// TIA Portal V18 export
VAR_GLOBAL   // PLC tag table "Default tag table"
   "AI11.01.01" AT %IW64 : Int;   // AHU NF Перепад тиску повітря (2.40)
   "AI11.01.02" AT %IW66 : Int;   // HS Вихід нагрівача (10.11)
   "DI11.01.01" AT %I0.0 : Bool;   // HS Режим роботи "Зима"
   "DI11.01.02" AT %I0.1 : Bool;   // HS Режим роботи "Авто"
   "DI11.01.03" AT %I0.2 : Bool;   // HS Відмова Котел 1
   "DI11.01.04" AT %I0.3 : Bool;   // HS Відмова Котел 2
   "DI11.01.05" AT %I0.4 : Bool;   // HS Норм. рівень води Котел 1 (10.80)
   "DI11.01.06" AT %I0.5 : Bool;   // HS Низький тиск Котел 1 (10.71)
   "DI11.01.07" AT %I0.6 : Bool;   // HS Високий тиск Котел 1 (10.72)
   "DI11.01.08" AT %I0.7 : Bool;   // HS Норм. рівень води Котел 2 (10.81)
   "DI11.01.09" AT %I1.0 : Bool;   // HS Низький тиск Котел 1 (10.73)
   "DI11.01.10" AT %I1.1 : Bool;   // HS Високий тиск Котел 1 (10.74)
   "DI11.01.11" AT %I1.2 : Bool;
   "DI11.01.12" AT %I1.3 : Bool;
   "DI11.01.13" AT %I1.4 : Bool;
   "DI11.01.14" AT %I1.5 : Bool;
   "DO11.01.01" AT %Q0.0 : Bool;
   "DO11.01.02" AT %Q0.1 : Bool;
   "DO11.01.03" AT %Q0.2 : Bool;
   "DO11.01.04" AT %Q0.3 : Bool;
   "DO11.01.05" AT %Q0.4 : Bool;
   "DO11.01.06" AT %Q0.5 : Bool;
   "DO11.01.07" AT %Q0.6 : Bool;
   "DO11.01.08" AT %Q0.7 : Bool;
   "DO11.01.09" AT %Q1.0 : Bool;
   "DO11.01.10" AT %Q1.1 : Bool;
   "AI11.02.01" AT %IW68 : Int;
   "AI11.02.02" AT %IW70 : Int;
   "AI11.02.03" AT %IW72 : Int;
   "AI11.02.04" AT %IW74 : Int;
   "AI11.02.05" AT %IW76 : Int;
   "AI11.02.06" AT %IW78 : Int;
   "AI11.02.07" AT %IW80 : Int;
   "AI11.02.08" AT %IW82 : Int;
   "AO11.03.01" AT %QW64 : Int;
   "AO11.03.02" AT %QW66 : Int;
   "AO11.03.03" AT %QW68 : Int;
   "AO11.03.04" AT %QW70 : Int;
   "DI11.04.01" AT %I2.0 : Bool;
   "DI11.04.02" AT %I2.1 : Bool;
   "DI11.04.03" AT %I2.2 : Bool;
   "DI11.04.04" AT %I2.3 : Bool;
   "DI11.04.05" AT %I2.4 : Bool;
   "DI11.04.06" AT %I2.5 : Bool;
   "DI11.04.07" AT %I2.6 : Bool;
   "DI11.04.08" AT %I2.7 : Bool;
   "DI11.04.09" AT %I3.0 : Bool;
   "DI11.04.10" AT %I3.1 : Bool;
   "DI11.04.11" AT %I3.2 : Bool;
   "DI11.04.12" AT %I3.3 : Bool;
   "DI11.04.13" AT %I3.4 : Bool;
   "DI11.04.14" AT %I3.5 : Bool;
   "DI11.04.15" AT %I3.6 : Bool;
   "DI11.04.16" AT %I3.7 : Bool;
   "DI11.05.01" AT %I4.0 : Bool;
   "DI11.05.02" AT %I4.1 : Bool;
   "DI11.05.03" AT %I4.2 : Bool;
   "DI11.05.04" AT %I4.3 : Bool;
   "DI11.05.05" AT %I4.4 : Bool;
   "DI11.05.06" AT %I4.5 : Bool;
   "DI11.05.07" AT %I4.6 : Bool;
   "DI11.05.08" AT %I4.7 : Bool;
   "DI11.05.09" AT %I5.0 : Bool;
   "DI11.05.10" AT %I5.1 : Bool;
   "DI11.05.11" AT %I5.2 : Bool;
   "DI11.05.12" AT %I5.3 : Bool;
   "DI11.05.13" AT %I5.4 : Bool;
   "DI11.05.14" AT %I5.5 : Bool;
   "DI11.05.15" AT %I5.6 : Bool;
   "DI11.05.16" AT %I5.7 : Bool;
   "DI11.06.01" AT %I6.0 : Bool;
   "DI11.06.02" AT %I6.1 : Bool;
   "DI11.06.03" AT %I6.2 : Bool;
   "DI11.06.04" AT %I6.3 : Bool;
   "DI11.06.05" AT %I6.4 : Bool;
   "DI11.06.06" AT %I6.5 : Bool;
   "DI11.06.07" AT %I6.6 : Bool;
   "DI11.06.08" AT %I6.7 : Bool;
   "DI11.06.09" AT %I7.0 : Bool;
   "DI11.06.10" AT %I7.1 : Bool;
   "DI11.06.11" AT %I7.2 : Bool;
   "DI11.06.12" AT %I7.3 : Bool;
   "DI11.06.13" AT %I7.4 : Bool;
   "DI11.06.14" AT %I7.5 : Bool;
   "DI11.06.15" AT %I7.6 : Bool;
   "DI11.06.16" AT %I7.7 : Bool;
   "DI11.07.01" AT %I8.0 : Bool;
   "DI11.07.02" AT %I8.1 : Bool;
   "DI11.07.03" AT %I8.2 : Bool;
   "DI11.07.04" AT %I8.3 : Bool;
   "DI11.07.05" AT %I8.4 : Bool;
   "DI11.07.06" AT %I8.5 : Bool;
   "DI11.07.07" AT %I8.6 : Bool;
   "DI11.07.08" AT %I8.7 : Bool;
   "DI11.07.09" AT %I9.0 : Bool;
   "DI11.07.10" AT %I9.1 : Bool;
   "DI11.07.11" AT %I9.2 : Bool;
   "DI11.07.12" AT %I9.3 : Bool;
   "DI11.07.13" AT %I9.4 : Bool;
   "DI11.07.14" AT %I9.5 : Bool;
   "DI11.07.15" AT %I9.6 : Bool;
   "DI11.07.16" AT %I9.7 : Bool;
   "DO11.08.01" AT %Q2.0 : Bool;
   "DO11.08.02" AT %Q2.1 : Bool;
   "DO11.08.03" AT %Q2.2 : Bool;
   "DO11.08.04" AT %Q2.3 : Bool;
   "DO11.08.05" AT %Q2.4 : Bool;
   "DO11.08.06" AT %Q2.5 : Bool;
   "DO11.08.07" AT %Q2.6 : Bool;
   "DO11.08.08" AT %Q2.7 : Bool;
   "DO11.08.09" AT %Q3.0 : Bool;
   "DO11.08.10" AT %Q3.1 : Bool;
   "DO11.08.11" AT %Q3.2 : Bool;
   "DO11.08.12" AT %Q3.3 : Bool;
   "DO11.08.13" AT %Q3.4 : Bool;
   "DO11.08.14" AT %Q3.5 : Bool;
   "DO11.08.15" AT %Q3.6 : Bool;
   "DO11.08.16" AT %Q3.7 : Bool;
   "DO11.09.01" AT %Q4.0 : Bool;
   "DO11.09.02" AT %Q4.1 : Bool;
   "DO11.09.03" AT %Q4.2 : Bool;
   "DO11.09.04" AT %Q4.3 : Bool;
   "DO11.09.05" AT %Q4.4 : Bool;
   "DO11.09.06" AT %Q4.5 : Bool;
   "DO11.09.07" AT %Q4.6 : Bool;
   "DO11.09.08" AT %Q4.7 : Bool;
   "DO11.09.09" AT %Q5.0 : Bool;
   "DO11.09.10" AT %Q5.1 : Bool;
   "DO11.09.11" AT %Q5.2 : Bool;
   "DO11.09.12" AT %Q5.3 : Bool;
   "DO11.09.13" AT %Q5.4 : Bool;
   "DO11.09.14" AT %Q5.5 : Bool;
   "DO11.09.15" AT %Q5.6 : Bool;
   "DO11.09.16" AT %Q5.7 : Bool;
   "AI11.10.01" AT %IW84 : Int;
   "AI11.10.02" AT %IW86 : Int;
   "AI11.10.03" AT %IW88 : Int;
   "AI11.10.04" AT %IW90 : Int;
   "AI11.10.05" AT %IW92 : Int;
   "AI11.10.06" AT %IW94 : Int;
   "AI11.10.07" AT %IW96 : Int;
   "AI11.10.08" AT %IW98 : Int;
   "AO11.11.01" AT %QW72 : Int;
   "AO11.11.02" AT %QW74 : Int;
   "AO11.11.03" AT %QW76 : Int;
   "AO11.11.04" AT %QW78 : Int;
END_VAR
